// TIA Portal V17 export
// export: Created 2026-10-01T22:10:23.5391934Z, ExportSetting WithDefaults, DisplayName Totally Integrated Automation Portal, DisplayVersion V17, DisplayName TIA Portal Openness, DisplayVersion V17, DisplayName TIA Portal Version Control Interface, DisplayVersion V17, DisplayName SINAMICS Startdrive Advanced, DisplayVersion V17, DisplayName SINAMICS Startdrive G130, G150, S120, S150, SINAMICS MV, G220, S200, S210, DisplayVersion V17, DisplayName SINAMICS Startdrive G110M, G120, G120C, G120D, G120P, G115D, DisplayVersion V17, DisplayName STEP 7 Professional, DisplayVersion V17, DisplayName STEP 7 Safety, DisplayVersion V17, DisplayName WinCC Basic/Comfort/Advanced, DisplayVersion V17, DisplayName WinCC Unified, DisplayVersion V17
FUNCTION_BLOCK "ZZ_LadTest_Sr"   // FB30, LAD
{ S7_Optimized_Access := 'TRUE' }
VERSION : 0.1
// stored: AutoNumber true, IsIECCheckEnabled false, IsRetainMemResEnabled false, MemoryReserve 100, SetENOAutomatically false, UDAEnableTagReadback false
   VAR_INPUT
      S : Bool;
      R : Bool;
   END_VAR
   VAR_OUTPUT
      Q1 : Bool;
      Q2 : Bool;
   END_VAR
   VAR
      Mem1 : Bool;
      Mem2 : Bool;
   END_VAR
BEGIN

REGION Network 1
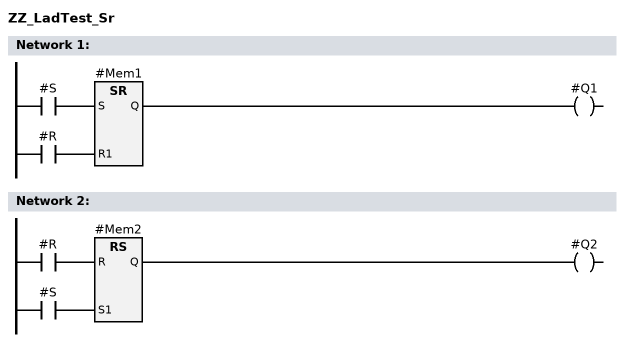
   RUNG wire#powerrail
      Contact( #S )
      S_SR(operand := #Mem1, r1 := wire#w1)
      Coil( #Q1 )
   END_RUNG
   RUNG wire#powerrail
      Contact( #R )
   END_RUNG wire#w1
   // the same network as SCL:
   IF #S THEN
       #Mem1 := TRUE;   // SR flip-flop
   END_IF;
   IF #R THEN #Mem1 := FALSE; END_IF;
   #Q1 := #Mem1;
END_REGION

REGION Network 2
   RUNG wire#powerrail
      Contact( #R )
      S_RS(operand := #Mem2, s1 := wire#w1)
      Coil( #Q2 )
   END_RUNG
   RUNG wire#powerrail
      Contact( #S )
   END_RUNG wire#w1
   // the same network as SCL:
   IF #R THEN
       #Mem2 := FALSE;   // RS flip-flop
   END_IF;
   IF #S THEN #Mem2 := TRUE; END_IF;
   #Q2 := #Mem2;
END_REGION
END_FUNCTION_BLOCK
